FUNCTION_BLOCK Mode_HMI (* Service Interface Function Block Type *)
  (* Standard: 61499-2 *)
  (* Version 0.0, 19/05/2022, SESA371406, Schneider Electric, template *)
  PACKAGE SE.Nereda;
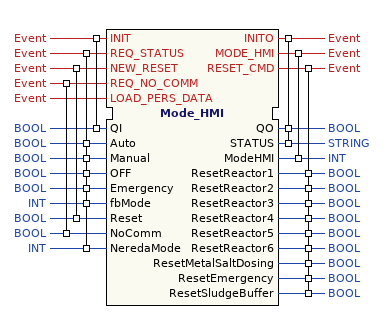
  EVENT_INPUT
    INIT WITH QI;
    REQ_STATUS WITH Auto, Manual, OFF, Emergency, fbMode, NeredaMode;
    NEW_RESET WITH Reset;
    REQ_NO_COMM WITH NoComm;
    LOAD_PERS_DATA;
  END_EVENT
  EVENT_OUTPUT
    INITO WITH QO, STATUS;
    MODE_HMI WITH ModeHMI;
    RESET_CMD WITH ResetReactor1, ResetReactor2, ResetReactor3, ResetReactor4, ResetReactor5, ResetReactor6, ResetMetalSaltDosing, ResetEmergency, ResetSludgeBuffer;
  END_EVENT
  VAR_INPUT
    QI : BOOL;
    Auto : BOOL;
    Manual : BOOL;
    OFF : BOOL;
    Emergency : BOOL;
    fbMode : INT;
    Reset : BOOL;
    NoComm : BOOL;
    NeredaMode : INT;
  END_VAR
  VAR_OUTPUT
    QO : BOOL; (* Event Output Qualifier *)
    STATUS : STRING; (* Service Status *)
    ModeHMI : INT;
    ResetReactor1 : BOOL;
    ResetReactor2 : BOOL;
    ResetReactor3 : BOOL;
    ResetReactor4 : BOOL;
    ResetReactor5 : BOOL;
    ResetReactor6 : BOOL;
    ResetMetalSaltDosing : BOOL;
    ResetEmergency : BOOL;
    ResetSludgeBuffer : BOOL;
  END_VAR
  SERVICE /
    SEQUENCE 
    END_SEQUENCE
  END_SERVICE
END_FUNCTION_BLOCK
